ABB RobotStudio station: Step_suction_gripper_20200824-193747.rsstn

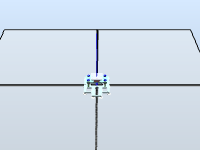
Station Station (saved by RobotStudio 6.8.8307.1040)
Layout (positions relative to the parent item):
  - Chwytak 1 [graphiccomponentgroup, from Diseño de proyecto\Suction_gripper.rslib]
    - NULL [graphiccomponentgroup, from Diseño de proyecto\Suction_gripper.rslib] at (-30.75, 147.99, -17.5) mm, rotated rx 90 ry 0 rz 0 deg
      - NULL [part, from Diseño de proyecto\Suction_gripper.rslib]
      - NULL [part, from Diseño de proyecto\Suction_gripper.rslib]
      - NULL [part, from Diseño de proyecto\Suction_gripper.rslib]
    - NULL [graphiccomponentgroup, from Diseño de proyecto\Suction_gripper.rslib] at (34.58, 147.99, -17.5) mm, rotated rx 90 ry 0 rz 0 deg
      - NULL [part, from Diseño de proyecto\Suction_gripper.rslib]
      - NULL [part, from Diseño de proyecto\Suction_gripper.rslib]
      - NULL [part, from Diseño de proyecto\Suction_gripper.rslib]
    - NULL [graphiccomponentgroup, from Diseño de proyecto\Suction_gripper.rslib] at (34.58, 54.52, -17.5) mm, rotated rx 90 ry 0 rz 0 deg
      - NULL [part, from Diseño de proyecto\Suction_gripper.rslib]
      - NULL [part, from Diseño de proyecto\Suction_gripper.rslib]
      - NULL [part, from Diseño de proyecto\Suction_gripper.rslib]
    - NULL [graphiccomponentgroup, from Diseño de proyecto\Suction_gripper.rslib] at (-30.75, 54.52, -17.5) mm, rotated rx 90 ry 0 rz 0 deg
      - NULL [part, from Diseño de proyecto\Suction_gripper.rslib]
      - NULL [part, from Diseño de proyecto\Suction_gripper.rslib]
      - NULL [part, from Diseño de proyecto\Suction_gripper.rslib]
    - NULL [graphiccomponentgroup, from Diseño de proyecto\Suction_gripper.rslib] at (-98.6, 101.25, -17.5) mm, rotated rx 90 ry 0 rz 0 deg
      - NULL [part, from Diseño de proyecto\Suction_gripper.rslib]
      - NULL [part, from Diseño de proyecto\Suction_gripper.rslib]
      - NULL [part, from Diseño de proyecto\Suction_gripper.rslib]
    - NULL [graphiccomponentgroup, from Diseño de proyecto\Suction_gripper.rslib] at (-30.75, -147.99, -17.5) mm, rotated rx 90 ry 0 rz 0 deg
      - NULL [part, from Diseño de proyecto\Suction_gripper.rslib]
      - NULL [part, from Diseño de proyecto\Suction_gripper.rslib]
      - NULL [part, from Diseño de proyecto\Suction_gripper.rslib]
    - NULL [graphiccomponentgroup, from Diseño de proyecto\Suction_gripper.rslib] at (34.58, -147.99, -17.5) mm, rotated rx 90 ry 0 rz 0 deg
      - NULL [part, from Diseño de proyecto\Suction_gripper.rslib]
      - NULL [part, from Diseño de proyecto\Suction_gripper.rslib]
      - NULL [part, from Diseño de proyecto\Suction_gripper.rslib]
    - NULL [graphiccomponentgroup, from Diseño de proyecto\Suction_gripper.rslib] at (34.58, -54.52, -17.5) mm, rotated rx 90 ry 0 rz 0 deg
      - NULL [part, from Diseño de proyecto\Suction_gripper.rslib]
      - NULL [part, from Diseño de proyecto\Suction_gripper.rslib]
      - NULL [part, from Diseño de proyecto\Suction_gripper.rslib]
    - NULL [graphiccomponentgroup, from Diseño de proyecto\Suction_gripper.rslib] at (100.63, -7.79, -17.5) mm, rotated rx 90 ry 0 rz 0 deg
      - NULL [part, from Diseño de proyecto\Suction_gripper.rslib]
      - NULL [part, from Diseño de proyecto\Suction_gripper.rslib]
      - NULL [part, from Diseño de proyecto\Suction_gripper.rslib]
    - NULL [graphiccomponentgroup, from Diseño de proyecto\Suction_gripper.rslib] at (100.63, -101.25, -17.5) mm, rotated rx 90 ry 0 rz 0 deg
      - NULL [part, from Diseño de proyecto\Suction_gripper.rslib]
      - NULL [part, from Diseño de proyecto\Suction_gripper.rslib]
      - NULL [part, from Diseño de proyecto\Suction_gripper.rslib]
    - NULL [graphiccomponentgroup, from Diseño de proyecto\Suction_gripper.rslib] at (100.63, 101.25, -17.5) mm, rotated rx 90 ry 0 rz 0 deg
      - NULL [part, from Diseño de proyecto\Suction_gripper.rslib]
      - NULL [part, from Diseño de proyecto\Suction_gripper.rslib]
      - NULL [part, from Diseño de proyecto\Suction_gripper.rslib]
    - NULL [graphiccomponentgroup, from Diseño de proyecto\Suction_gripper.rslib] at (-30.75, -54.52, -17.5) mm, rotated rx 90 ry 0 rz 0 deg
      - NULL [part, from Diseño de proyecto\Suction_gripper.rslib]
      - NULL [part, from Diseño de proyecto\Suction_gripper.rslib]
      - NULL [part, from Diseño de proyecto\Suction_gripper.rslib]
    - NULL [graphiccomponentgroup, from Diseño de proyecto\Suction_gripper.rslib] at (-98.6, -101.25, -17.5) mm, rotated rx 90 ry 0 rz 0 deg
      - NULL [part, from Diseño de proyecto\Suction_gripper.rslib]
      - NULL [part, from Diseño de proyecto\Suction_gripper.rslib]
      - NULL [part, from Diseño de proyecto\Suction_gripper.rslib]
    - NULL [graphiccomponentgroup, from Diseño de proyecto\Suction_gripper.rslib] at (-98.6, -7.79, -17.5) mm, rotated rx 90 ry 0 rz 0 deg
      - NULL [part, from Diseño de proyecto\Suction_gripper.rslib]
      - NULL [part, from Diseño de proyecto\Suction_gripper.rslib]
      - NULL [part, from Diseño de proyecto\Suction_gripper.rslib]
    - NULL [part, from Diseño de proyecto\Suction_gripper.rslib]
    - NULL [part, from Diseño de proyecto\Suction_gripper.rslib] at (0, 0, 61.15) mm
    - NULL [part, from Diseño de proyecto\Suction_gripper.rslib] at (70, -33, 75) mm, rotated rx 0 ry 90 rz 0 deg
    - NULL [part, from Diseño de proyecto\Suction_gripper.rslib] at (-70, -33, 43) mm, rotated rx 0 ry -90 rz 0 deg
    - NULL [part, from Diseño de proyecto\Suction_gripper.rslib] at (70, 33, 75) mm, rotated rx 0 ry 90 rz 0 deg
    - NULL [part, from Diseño de proyecto\Suction_gripper.rslib] at (-70, 33, 75) mm, rotated rx 0 ry 90 rz 0 deg
    - NULL [part, from Diseño de proyecto\Suction_gripper.rslib] at (70, -33, 75) mm, rotated rx 180 ry 0 rz -157.48 deg
    - NULL [part, from Diseño de proyecto\Suction_gripper.rslib] at (70, 33, 75) mm, rotated rx 180 ry 0 rz -157.48 deg
    - NULL [part, from Diseño de proyecto\Suction_gripper.rslib] at (-70, 33, 10) mm
    - NULL [part, from Diseño de proyecto\Suction_gripper.rslib] at (-70, -33, 10) mm, rotated rx 0 ry 0 rz -10.23 deg
    - NULL [part, from Diseño de proyecto\Suction_gripper.rslib] at (0, 0, 69.15) mm
    - NULL [part, from Diseño de proyecto\Suction_gripper.rslib] at (64, 0, 62.15) mm, rotated rx 180 ry 0 rz -157.48 deg
    - NULL [part, from Diseño de proyecto\Suction_gripper.rslib] at (-64, 0, 62.15) mm, rotated rx 180 ry 0 rz -157.48 deg
    - NULL [part, from Diseño de proyecto\Suction_gripper.rslib] at (64, 0, 10) mm
    - NULL [part, from Diseño de proyecto\Suction_gripper.rslib] at (-64, 0, 10) mm
    - NULL [part, from Diseño de proyecto\Suction_gripper.rslib] at (0, 0, 92.15) mm, rotated rx 180 ry 0 rz 180 deg
    - NULL [part, from Diseño de proyecto\Suction_gripper.rslib] at (70, 33, 61.15) mm, rotated rx 180 ry 0 rz -157.48 deg
    - NULL [part, from Diseño de proyecto\Suction_gripper.rslib] at (-70, 33, 61.15) mm, rotated rx 180 ry 0 rz -157.48 deg
    - NULL [part, from Diseño de proyecto\Suction_gripper.rslib] at (70, -33, 61.15) mm, rotated rx 180 ry 0 rz -157.48 deg
    - NULL [part, from Diseño de proyecto\Suction_gripper.rslib] at (-70, -33, 61.15) mm, rotated rx 180 ry 0 rz -157.48 deg
    - NULL [part, from Diseño de proyecto\Suction_gripper.rslib] at (70, -33, 75) mm
    - NULL [part, from Diseño de proyecto\Suction_gripper.rslib] at (-70, 33, 75) mm, rotated rx 0 ry 0 rz 22.23 deg
    - NULL [part, from Diseño de proyecto\Suction_gripper.rslib] at (-70, -33, 75) mm
    - NULL [part, from Diseño de proyecto\Suction_gripper.rslib] at (70, 33, 75) mm
    - NULL [part, from Diseño de proyecto\Suction_gripper.rslib] at (63.98, 0.08, 58.7) mm
    - NULL [part, from Diseño de proyecto\Suction_gripper.rslib] at (-64.1, -0.17, 58.7) mm
